// TIA Portal V21 export
DATA_BLOCK "AMEND"   // DB36
{ S7_Optimized_Access := 'FALSE' }
   VAR
      "PRODUCT NAME" : String[80] := '$L$RPRODUCT NAME        :';
      "BATCH NO" : String[80] := '$L$RBATCH NO            :';
      "OPERATOR NAME" : String[80] := '$L$ROPERATOR NAME       :UDAYLAL';
      "RECIPE TYPE" : String[80] := '$L$R        :';
      "EQUIPMENT ID" : String[80] := '$L$REQUIPMENT ID        :C1/A/INJ/AUT-05';
      "OP PRODUCT NAME" : String[80] := '';
      "TUNNEL MODE" : String[80] := '$L$RPROCESS                    :    NONE';
      CIP : String[30] := 'CLOSURE CYCLE SELECTED';
      STANDARD1 : String[30] := 'STANDARD1 CYCLE SELECTED';
      STANDARD2 : String[30] := 'STANDARD2 CYCLE SELECTED';
      BOWIE : String[30] := 'BOWIE DICK CYCLE SELECTED';
      NONE : String[30] := 'NONE';
      "BATCH SIZE" : String[80] := '  CYCLE NO            :0488';
      "CONTAINER SIZE" : String[80] := '  CONTAINER SIZE      :';
      HPHV : String[80] := 'HPHV CYCLE SELECTED';
      LEAK : String[80] := 'VACUUM LEAK TEST SELECTED';
      start : String[80] := '46';
      end : String[80] := '18:52:46';
      "END PV" : String[80] := '  18:52:46    0.086     48.4    103.2     92.2     93.1    105.8 ';
      "PRINT PV" : String[80] := '$L$R18:52:46    0.086     48.4    103.2     92.2     93.1    105.8  NOT START';
      "PRINT CYCLE ABORT" : String[80] := '18:52:19   ******CYCLE ABORTED******     ';
      QUANTITY : String[80] := '  ';
   END_VAR
BEGIN
END_DATA_BLOCK
